PROGRAM OmronServoEnable
VAR
END_VAR

IF PowerOnDelay.Q AND NOT EmergencyStop THEN
	ARwDO[eY10007_STN09SLOWPULLMECHANISMSERVOMOTOR_ERRORSTOP].00 := TRUE;
	ARwDO[eY10008_Arm01HorizontalServoMotor_ErrorStop].00 := TRUE;
	ARwDO[eY10009_Arm01VerticalServoMotor_ErrorStop].00 := TRUE;
	ELSE
	ARwDO[eY10007_STN09SLOWPULLMECHANISMSERVOMOTOR_ERRORSTOP].00 := FALSE;
	ARwDO[eY10008_Arm01HorizontalServoMotor_ErrorStop].00 := FALSE;
	ARwDO[eY10009_Arm01VerticalServoMotor_ErrorStop].00 := FALSE;
END_IF

END_PROGRAM

(* stored: Version 1.1.0.1, ProductVersion 3.1.4024.12
   POU OmronServoEnable: Id {c8aa9bd6-7f3d-431d-9123-154fdcefa32f}, SpecialFunc None *)
